Staubli VAL3: getAnaValue.pgx

public program getAnaValue(num& x_nValue[], num x_nIndex)
begin
  x_nValue=aioGet(saveInOut:aio_out[x_nIndex])
end
